% RSLogix 500 project ALARM & FAULT_DETECTION_BAK000.RSS, saved by version 8.30.00.16 %
PROJECT "TANK_A&F"    % processor: Bul.1763 MicroLogix 1100 Series B %

PROGRAM FILES
  LAD 2 "SYSTEM"  5 rungs
  LAD 3 "IN/OUT"  6 rungs
  LAD 4 "MAIN"  3 rungs
  LAD 5 "ALARM"  7 rungs
  LAD 6 "FAULT"  6 rungs

DATA FILES
  O0 OUTPUT  4 elements
  I1 INPUT  6 elements
  S2 STATUS  66 elements
  B3 BINARY  100 elements
  T4 TIMER  4 elements
  C5 COUNTER  1 elements
  R6 CONTROL  1 elements
  N7 INTEGER  1 elements
  F8 FLOAT  1 elements

LADDER 2 "SYSTEM"
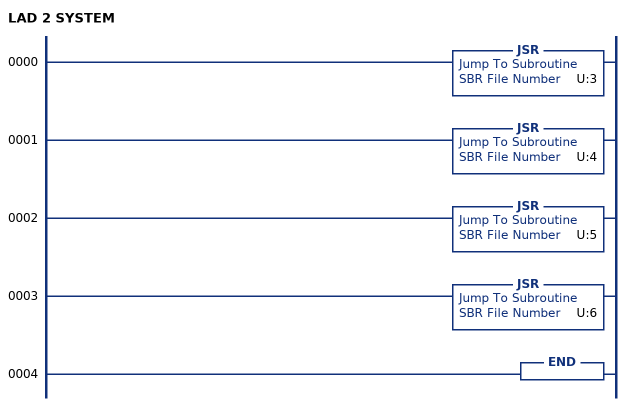
% Rung: 0 %
SOR JSR U:3 EOR
% Rung: 1 %
SOR JSR U:4 EOR
% Rung: 2 %
SOR JSR U:5 EOR
% Rung: 3 %
SOR JSR U:6 EOR
% Rung: 4 %
SOR END EOR

LADDER 3 "IN/OUT"
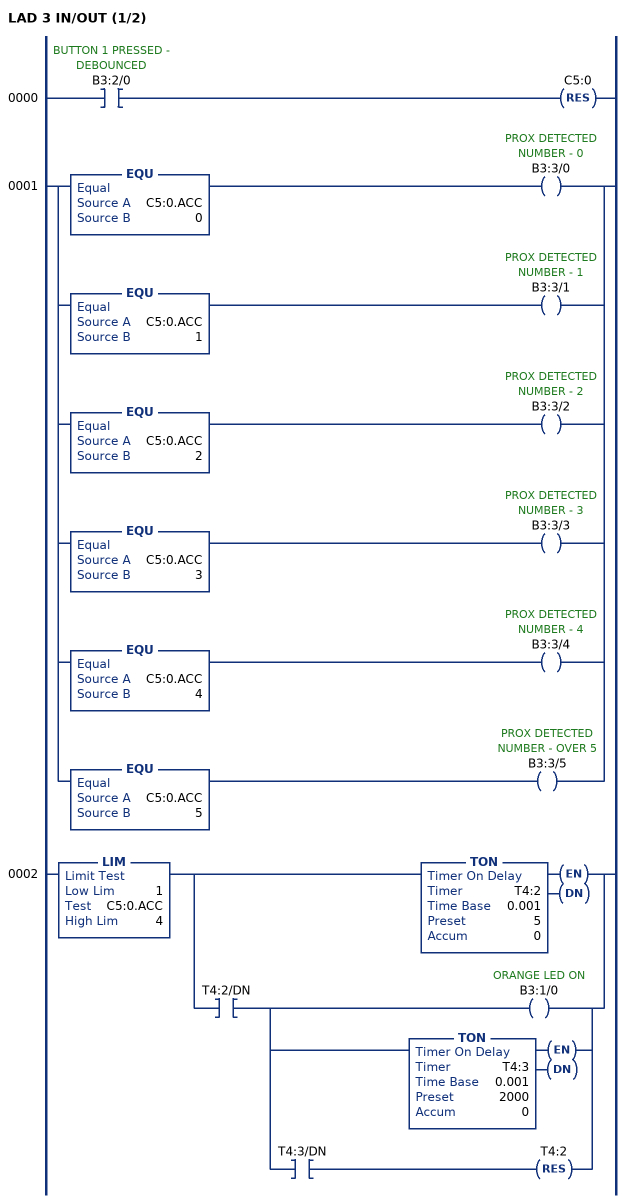
% Rung: 0 %
SOR XIC B3:2/0 RES C5:0 EOR
%   B3:2/0  "BUTTON 1 PRESSED - DEBOUNCED" %
% Rung: 1 %
SOR BST EQU C5:0.ACC 0 OTE B3:3/0 NXB EQU C5:0.ACC 1 OTE B3:3/1 NXB EQU C5:0.ACC 2 OTE B3:3/2 NXB EQU C5:0.ACC 3 OTE B3:3/3 NXB EQU C5:0.ACC 4 OTE B3:3/4 NXB EQU C5:0.ACC 5 OTE B3:3/5 BND EOR
%   B3:3/0  "PROX DETECTED NUMBER - 0" %
%   B3:3/1  "PROX DETECTED NUMBER - 1" %
%   B3:3/2  "PROX DETECTED NUMBER - 2" %
%   B3:3/3  "PROX DETECTED NUMBER - 3" %
%   B3:3/4  "PROX DETECTED NUMBER - 4" %
%   B3:3/5  "PROX DETECTED NUMBER - OVER 5" %
% Rung: 2 %
SOR LIM 1 C5:0.ACC 4 BST TON T4:2 0.001 5 0 NXB XIC T4:2/DN BST OTE B3:1/0 NXB TON T4:3 0.001 2000 0 NXB XIC T4:3/DN RES T4:2 BND BND EOR
%   B3:1/0  "ORANGE LED ON" %

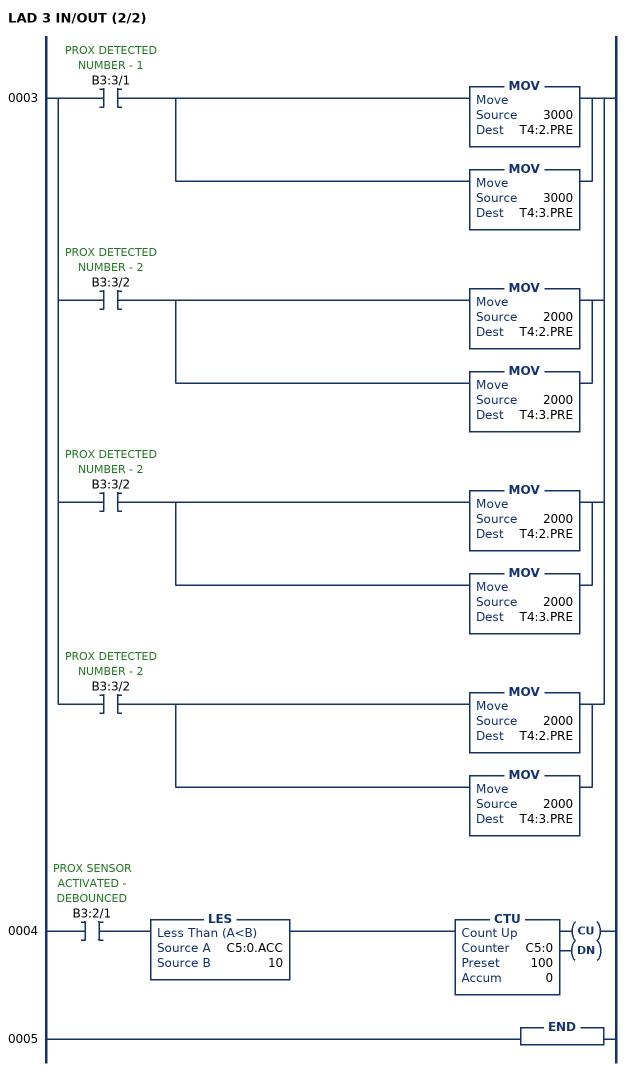
% Rung: 3 %
SOR BST XIC B3:3/1 BST MOV 3000 T4:2.PRE NXB MOV 3000 T4:3.PRE BND NXB XIC B3:3/2 BST MOV 2000 T4:2.PRE NXB MOV 2000 T4:3.PRE BND NXB XIC B3:3/2 BST MOV 2000 T4:2.PRE NXB MOV 2000 T4:3.PRE BND NXB XIC B3:3/2 BST MOV 2000 T4:2.PRE NXB MOV 2000 T4:3.PRE BND BND EOR
%   B3:3/1  "PROX DETECTED NUMBER - 1" %
%   B3:3/2  "PROX DETECTED NUMBER - 2" %
% Rung: 4 %
SOR XIC B3:2/1 LES C5:0.ACC 10 CTU C5:0 100 0 EOR
%   B3:2/1  "PROX SENSOR ACTIVATED - DEBOUNCED" %
% Rung: 5 %
SOR END EOR

LADDER 4 "MAIN"
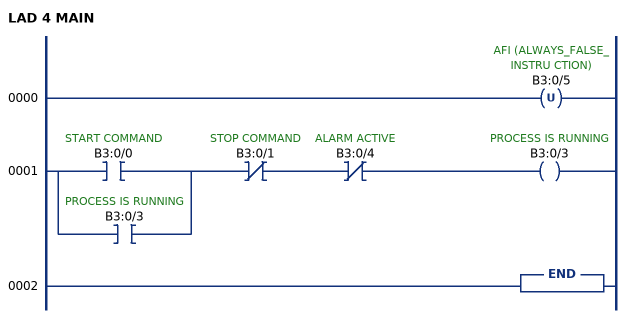
% Rung: 0 %
SOR OTU B3:0/5 EOR
%   B3:0/5  "AFI (ALWAYS_FALSE_INSTRU CTION)" %
% Rung: 1 %
SOR BST XIC B3:0/0 NXB XIC B3:0/3 BND XIO B3:0/1 XIO B3:0/4 OTE B3:0/3 EOR
%   B3:0/0  "START COMMAND" %
%   B3:0/3  "PROCESS IS RUNNING" %
%   B3:0/1  "STOP COMMAND" %
%   B3:0/4  "ALARM ACTIVE" %
% Rung: 2 %
SOR END EOR

LADDER 5 "ALARM"
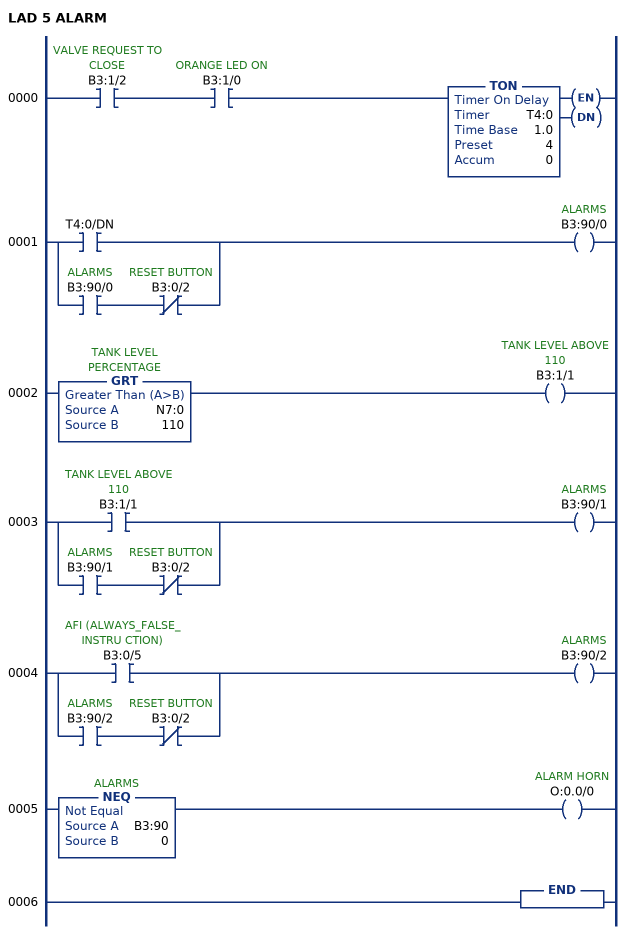
% Rung: 0 %
SOR XIC B3:1/2 XIC B3:1/0 TON T4:0 1.0 4 0 EOR
%   B3:1/2  "VALVE REQUEST TO CLOSE" %
%   B3:1/0  "ORANGE LED ON" %
% Rung: 1 %
SOR BST XIC T4:0/DN NXB XIC B3:90/0 XIO B3:0/2 BND OTE B3:90/0 EOR
%   B3:90/0  "ALARMS" %
%   B3:0/2  "RESET BUTTON" %
% Rung: 2 %
SOR GRT N7:0 110 OTE B3:1/1 EOR
%   N7:0  "TANK LEVEL PERCENTAGE" %
%   B3:1/1  "TANK LEVEL ABOVE 110" %
% Rung: 3 %
SOR BST XIC B3:1/1 NXB XIC B3:90/1 XIO B3:0/2 BND OTE B3:90/1 EOR
%   B3:1/1  "TANK LEVEL ABOVE 110" %
%   B3:90/1  "ALARMS" %
%   B3:0/2  "RESET BUTTON" %
% Rung: 4 %
SOR BST XIC B3:0/5 NXB XIC B3:90/2 XIO B3:0/2 BND OTE B3:90/2 EOR
%   B3:0/5  "AFI (ALWAYS_FALSE_INSTRU CTION)" %
%   B3:90/2  "ALARMS" %
%   B3:0/2  "RESET BUTTON" %
% Rung: 5 %
SOR NEQ B3:90 0 OTE O:0.0/0 EOR
%   B3:90  "ALARMS" %
%   O:0.0/0  "ALARM HORN" %
% Rung: 6 %
SOR END EOR

LADDER 6 "FAULT"
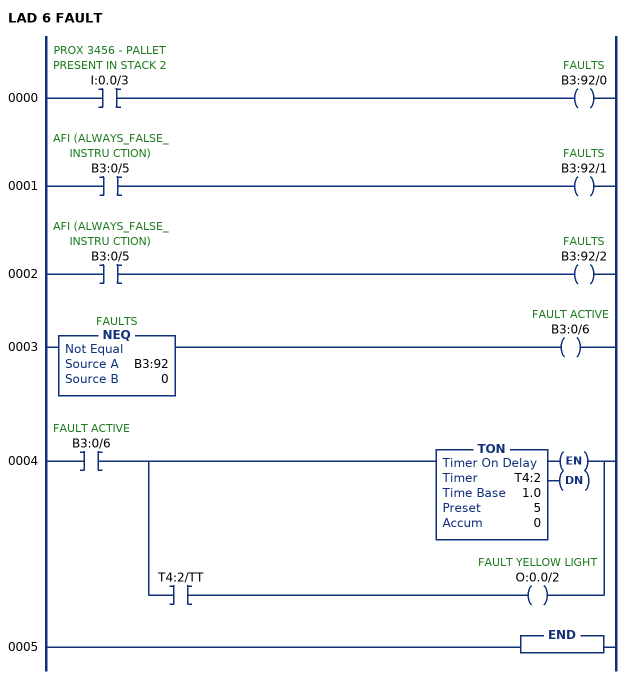
% Rung: 0 %
SOR XIC I:0.0/3 OTE B3:92/0 EOR
%   I:0.0/3  "PROX 3456 - PALLET PRESENT IN STACK 2" %
%   B3:92/0  "FAULTS" %
% Rung: 1 %
SOR XIC B3:0/5 OTE B3:92/1 EOR
%   B3:0/5  "AFI (ALWAYS_FALSE_INSTRU CTION)" %
%   B3:92/1  "FAULTS" %
% Rung: 2 %
SOR XIC B3:0/5 OTE B3:92/2 EOR
%   B3:0/5  "AFI (ALWAYS_FALSE_INSTRU CTION)" %
%   B3:92/2  "FAULTS" %
% Rung: 3 %
SOR NEQ B3:92 0 OTE B3:0/6 EOR
%   B3:92  FAULTS %
%   B3:0/6  "FAULT ACTIVE" %
% Rung: 4 %
SOR XIC B3:0/6 BST TON T4:2 1.0 5 0 NXB XIC T4:2/TT OTE O:0.0/2 BND EOR
%   B3:0/6  "FAULT ACTIVE" %
%   O:0.0/2  "FAULT YELLOW LIGHT" %
% Rung: 5 %
SOR END EOR

OTHER DOCUMENTED ADDRESSES
  B3:91  ALARMS_2
  O:0.0/1  "ALARM HORN"
  T4:1/TT  "ALARM HORN TIMER"

DATA TABLE (non-zero values as saved)
DATA T4
% .PRE .ACC %
% T4:0 % 4 0
% T4:1 % 5000 0
% T4:2 % 5 0
% T4:3 % 2000 0
DATA C5
% .PRE .ACC %
% C5:0 % 100 0
